  [744] = "0.00,0.00,0.00,90.00,0.00,90.00,0,"
  [745] = "0.00,0.00,0.00,90.00,0.00,90.00,0,"
  [746] = "0.00,0.00,0.00,90.00,0.00,90.00,0,"
  [747] = "0.00,0.00,0.00,90.00,0.00,90.00,1,"
  [748] = "0.00,0.00,0.00,90.00,0.00,90.00,0,"
  [749] = "0.00,0.00,0.00,90.00,0.00,90.00,0,"
  [750] = "0.00,0.00,0.00,90.00,0.00,90.00,0,"
  [751] = "0.00,0.00,0.00,90.00,0.00,90.00,1,"
  [752] = "0.00,0.00,0.00,90.00,0.00,90.00,0,"
  [753] = "0.00,0.00,0.00,90.00,0.00,90.00,0,"
  [754] = "0.00,0.00,0.00,90.00,0.00,90.00,0,"
  [755] = "0.00,0.00,0.00,90.00,0.00,90.00,1,"
  [756] = "0.00,0.00,0.00,90.00,0.00,90.00,0,"
  [757] = "0.00,0.00,0.00,90.00,0.00,90.00,0,"
  [758] = "0.00,0.00,0.00,90.00,0.00,90.00,0,"
  [759] = "0.00,0.00,0.00,90.00,0.00,90.00,1,"
  [760] = "0.00,0.00,0.00,90.00,0.00,90.00,0,"
  [761] = "0.00,0.00,0.00,90.00,0.00,90.00,0,"
  [762] = "0.00,0.00,0.00,90.00,0.00,90.00,0,"
  [763] = "0.00,0.00,0.00,90.00,0.00,90.00,1,"
  [764] = "0.00,0.00,0.00,90.00,0.00,90.00,0,"
  [765] = "0.00,0.00,0.00,90.00,0.00,90.00,0,"
  [766] = "0.00,0.00,0.00,90.00,0.00,90.00,0,"
  [767] = "0.00,0.00,0.00,90.00,0.00,90.00,1,"
  [768] = "0.00,0.00,0.00,90.00,0.00,90.00,0,"
  [769] = "0.00,0.00,0.00,90.00,0.00,90.00,0,"
  [770] = "0.00,0.00,0.00,90.00,0.00,90.00,0,"
  [771] = "0.00,0.00,0.00,90.00,0.00,90.00,1,"
  [772] = "0.00,0.00,0.00,90.00,0.00,90.00,0,"
  [773] = "0.00,0.00,0.00,90.00,0.00,90.00,0,"
  [774] = "0.00,0.00,0.00,90.00,0.00,90.00,0,"
  [775] = "0.00,0.00,0.00,90.00,0.00,90.00,1,"
  [776] = "0.00,0.00,0.00,90.00,0.00,90.00,0,"
  [777] = "0.00,0.00,0.00,90.00,0.00,90.00,0,"
  [778] = "0.00,0.00,0.00,90.00,0.00,90.00,0,"
  [779] = "0.00,0.00,0.00,90.00,0.00,90.00,1,"
  [780] = "0.00,0.00,0.00,90.00,0.00,90.00,0,"
  [781] = "0.00,0.00,0.00,90.00,0.00,90.00,0,"
  [782] = "0.00,0.00,0.00,90.00,0.00,90.00,0,"
  [783] = "0.00,0.00,0.00,90.00,0.00,90.00,1,"
  [784] = "0.00,0.00,0.00,90.00,0.00,90.00,0,"
  [785] = "0.00,0.00,0.00,90.00,0.00,90.00,0,"
  [786] = "0.00,0.00,0.00,90.00,0.00,90.00,0,"
  [787] = "0.00,0.00,0.00,90.00,0.00,90.00,1,"
  [788] = "0.00,0.00,0.00,90.00,0.00,90.00,0,"
  [789] = "0.00,0.00,0.00,90.00,0.00,90.00,0,"
  [790] = "0.00,0.00,0.00,90.00,0.00,90.00,0,"
  [791] = "0.00,0.00,0.00,90.00,0.00,90.00,1,"
  [792] = "0.00,0.00,0.00,90.00,0.00,90.00,0,"
  [793] = "0.00,0.00,0.00,90.00,0.00,90.00,0,"
  [794] = "0.00,0.00,0.00,90.00,0.00,90.00,0,"
  [795] = "0.00,0.00,0.00,90.00,0.00,90.00,1,"
  [796] = "0.00,0.00,0.00,90.00,0.00,90.00,0,"
  [797] = "0.00,0.00,0.00,90.00,0.00,90.00,0,"
  [798] = "0.00,0.00,0.00,90.00,0.00,90.00,0,"
  [799] = "0.00,0.00,0.00,90.00,0.00,90.00,1,"
  [800] = "0.00,0.00,0.00,90.00,0.00,90.00,0,"
  [801] = "0.00,0.00,0.00,90.00,0.00,90.00,0,"
  [802] = "0.00,0.00,0.00,90.00,0.00,90.00,0,"
  [803] = "0.00,0.00,0.00,90.00,0.00,90.00,1,"
  [804] = "0.00,0.00,0.00,90.00,0.00,90.00,0,"
  [805] = "0.00,0.00,0.00,90.00,0.00,90.00,0,"
  [806] = "0.00,0.00,0.00,90.00,0.00,90.00,0,"
  [807] = "0.00,0.00,0.00,90.00,0.00,90.00,1,"
  [808] = "0.00,0.00,0.00,90.00,0.00,90.00,0,"
  [809] = "0.00,0.00,0.00,90.00,0.00,90.00,0,"
  [810] = "0.00,0.00,0.00,90.00,0.00,90.00,0,"
  [811] = "0.00,0.00,0.00,90.00,0.00,90.00,1,"
  [812] = "0.00,0.00,0.00,90.00,0.00,90.00,0,"
  [813] = "0.00,0.00,0.00,90.00,0.00,90.00,0,"
  [814] = "0.00,0.00,0.00,90.00,0.00,90.00,0,"
  [815] = "0.00,0.00,0.00,90.00,0.00,90.00,1,"
  [816] = "0.00,0.00,0.00,90.00,0.00,90.00,0,"
  [817] = "0.00,0.00,0.00,90.00,0.00,90.00,0,"
  [818] = "0.00,0.00,0.00,90.00,0.00,90.00,0,"
  [819] = "0.00,0.00,0.00,90.00,0.00,90.00,1,"
  [820] = "0.00,0.00,0.00,90.00,0.00,90.00,0,"
  [821] = "0.00,0.00,0.00,90.00,0.00,90.00,0,"
  [822] = "0.00,0.00,0.00,90.00,0.00,90.00,0,"
  [823] = "0.00,0.00,0.00,90.00,0.00,90.00,1,"
  [824] = "0.00,0.00,0.00,90.00,0.00,90.00,0,"
  [825] = "0.00,0.00,0.00,90.00,0.00,90.00,0,"
  [826] = "0.00,0.00,0.00,90.00,0.00,90.00,0,"
  [827] = "0.00,0.00,0.00,90.00,0.00,90.00,1,"
  [828] = "0.00,0.00,0.00,90.00,0.00,90.00,0,"
  [829] = "0.00,0.00,0.00,90.00,0.00,90.00,0,"
  [830] = "0.00,0.00,0.00,90.00,0.00,90.00,0,"
  [831] = "0.00,0.00,0.00,90.00,0.00,90.00,1,"
  [832] = "0.00,0.00,0.00,90.00,0.00,90.00,0,"
  [833] = "0.00,0.00,0.00,90.00,0.00,90.00,0,"
  [834] = "0.00,0.00,0.00,90.00,0.00,90.00,0,"
  [835] = "0.00,0.00,0.00,90.00,0.00,90.00,1,"
  [836] = "0.00,0.00,0.00,90.00,0.00,90.00,0,"
  [837] = "0.00,0.00,0.00,90.00,0.00,90.00,0,"
  [838] = "0.00,0.00,0.00,90.00,0.00,90.00,0,"
  [839] = "0.00,0.00,0.00,90.00,0.00,90.00,1,"
  [840] = "0.00,0.00,0.00,90.00,0.00,90.00,0,"
  [841] = "0.00,0.00,0.00,90.00,0.00,90.00,0,"
  [842] = "0.00,0.00,0.00,90.00,0.00,90.00,0,"
  [843] = "0.00,0.00,0.00,90.00,0.00,90.00,1,"
  [844] = "0.00,0.00,0.00,90.00,0.00,90.00,0,"
  [845] = "0.00,0.00,0.00,90.00,0.00,90.00,0,"
  [846] = "0.00,0.00,0.00,90.00,0.00,90.00,0,"
  [847] = "0.00,0.00,0.00,90.00,0.00,90.00,1,"
  [848] = "0.00,0.00,0.00,90.00,0.00,90.00,0,"
  [849] = "0.00,0.00,0.00,90.00,0.00,90.00,0,"
  [850] = "0.00,0.00,0.00,90.00,0.00,90.00,0,"
  [851] = "0.00,0.00,0.00,90.00,0.00,90.00,1,"
  [852] = "0.00,0.00,0.00,90.00,0.00,90.00,0,"
  [853] = "0.00,0.00,0.00,90.00,0.00,90.00,0,"
  [854] = "0.00,0.00,0.00,90.00,0.00,90.00,0,"
  [855] = "0.00,0.00,0.00,90.00,0.00,90.00,1,"
  [856] = "0.00,0.00,0.00,90.00,0.00,90.00,0,"
  [857] = "0.00,0.00,0.00,90.00,0.00,90.00,0,"
  [858] = "0.00,0.00,0.00,90.00,0.00,90.00,0,"
  [859] = "0.00,0.00,0.00,90.00,0.00,90.00,1,"
  [860] = "0.00,0.00,0.00,90.00,0.00,90.00,0,"
  [861] = "0.00,0.00,0.00,90.00,0.00,90.00,0,"
  [862] = "0.00,0.00,0.00,90.00,0.00,90.00,0,"
  [863] = "0.00,0.00,0.00,90.00,0.00,90.00,1,"
  [864] = "0.00,0.00,0.00,90.00,0.00,90.00,0,"
  [865] = "0.00,0.00,0.00,90.00,0.00,90.00,0,"
  [866] = "0.00,0.00,0.00,90.00,0.00,90.00,0,"
  [867] = "0.00,0.00,0.00,90.00,0.00,90.00,1,"
  [868] = "0.00,0.00,0.00,90.00,0.00,90.00,0,"
  [869] = "0.00,0.00,0.00,90.00,0.00,90.00,0,"
  [870] = "0.00,0.00,0.00,90.00,0.00,90.00,0,"
  [871] = "0.00,0.00,0.00,90.00,0.00,90.00,1,"
  [872] = "0.00,0.00,0.00,90.00,0.00,90.00,0,"
  [873] = "0.00,0.00,0.00,90.00,0.00,90.00,0,"
  [874] = "0.00,0.00,0.00,90.00,0.00,90.00,0,"
  [875] = "0.00,0.00,0.00,90.00,0.00,90.00,1,"
  [876] = "0.00,0.00,0.00,90.00,0.00,90.00,0,"
  [877] = "0.00,0.00,0.00,90.00,0.00,90.00,0,"
  [878] = "0.00,0.00,0.00,90.00,0.00,90.00,0,"
  [879] = "0.00,0.00,0.00,90.00,0.00,90.00,1,"
  [880] = "0.00,0.00,0.00,90.00,0.00,90.00,0,"
  [881] = "0.00,0.00,0.00,90.00,0.00,90.00,0,"
  [882] = "0.00,0.00,0.00,90.00,0.00,90.00,0,"
  [883] = "0.00,0.00,0.00,90.00,0.00,90.00,1,"
  [884] = "0.00,0.00,0.00,90.00,0.00,90.00,0,"
  [885] = "0.00,0.00,0.00,90.00,0.00,90.00,0,"
  [886] = "0.00,0.00,0.00,90.00,0.00,90.00,0,"
  [887] = "0.00,0.00,0.00,90.00,0.00,90.00,1,"
  [888] = "0.00,0.00,0.00,90.00,0.00,90.00,0,"
  [889] = "0.00,0.00,0.00,90.00,0.00,90.00,0,"
  [890] = "0.00,0.00,0.00,90.00,0.00,90.00,0,"
  [891] = "0.00,0.00,0.00,90.00,0.00,90.00,1,"
  [892] = "0.00,0.00,0.00,90.00,0.00,90.00,0,"
  [893] = "0.00,0.00,0.00,90.00,0.00,90.00,0,"
  [894] = "0.00,0.00,0.00,90.00,0.00,90.00,0,"
  [895] = "0.00,0.00,0.00,90.00,0.00,90.00,1,"
  [896] = "0.00,0.00,0.00,90.00,0.00,90.00,0,"
  [897] = "0.00,0.00,0.00,90.00,0.00,90.00,0,"
  [898] = "0.00,0.00,0.00,90.00,0.00,90.00,0,"
  [899] = "0.00,0.00,0.00,90.00,0.00,90.00,1,"
  [900] = "0.00,0.00,0.00,90.00,0.00,90.00,0,"
  [901] = "0.00,0.00,0.00,90.00,0.00,90.00,0,"
  [902] = "0.00,0.00,0.00,90.00,0.00,90.00,0,"
  [903] = "0.00,0.00,0.00,90.00,0.00,90.00,1,"
  [904] = "0.00,0.00,0.00,90.00,0.00,90.00,0,"
  [905] = "0.00,0.00,0.00,90.00,0.00,90.00,0,"
  [906] = "0.00,0.00,0.00,90.00,0.00,90.00,0,"
  [907] = "0.00,0.00,0.00,90.00,0.00,90.00,1,"
  [908] = "0.00,0.00,0.00,90.00,0.00,90.00,0,"
  [909] = "0.00,0.00,0.00,90.00,0.00,90.00,0,"
  [910] = "0.00,0.00,0.00,90.00,0.00,90.00,0,"
  [911] = "0.00,0.00,0.00,90.00,0.00,90.00,1,"
  [912] = "0.00,0.00,0.00,90.00,0.00,90.00,0,"
  [913] = "0.00,0.00,0.00,90.00,0.00,90.00,0,"
  [914] = "0.00,0.00,0.00,90.00,0.00,90.00,0,"
  [915] = "0.00,0.00,0.00,90.00,0.00,90.00,1,"
  [916] = "0.00,0.00,0.00,90.00,0.00,90.00,0,"
  [917] = "0.00,0.00,0.00,90.00,0.00,90.00,0,"
  [918] = "0.00,0.00,0.00,90.00,0.00,90.00,0,"
  [919] = "0.00,0.00,0.00,90.00,0.00,90.00,1,"
  [920] = "0.00,0.00,0.00,90.00,0.00,90.00,0,"
  [921] = "0.00,0.00,0.00,90.00,0.00,90.00,0,"
  [922] = "0.00,0.00,0.00,90.00,0.00,90.00,0,"
  [923] = "0.00,0.00,0.00,90.00,0.00,90.00,1,"
  [924] = "0.00,0.00,0.00,90.00,0.00,90.00,0,"
  [925] = "0.00,0.00,0.00,90.00,0.00,90.00,0,"
  [926] = "0.00,0.00,0.00,90.00,0.00,90.00,0,"
  [927] = "0.00,0.00,0.00,90.00,0.00,90.00,1,"
  [928] = "0.00,0.00,0.00,90.00,0.00,90.00,0,"
  [929] = "0.00,0.00,0.00,90.00,0.00,90.00,0,"
  [930] = "0.00,0.00,0.00,90.00,0.00,90.00,0,"
  [931] = "0.00,0.00,0.00,90.00,0.00,90.00,1,"
  [932] = "0.00,0.00,0.00,90.00,0.00,90.00,0,"
  [933] = "0.00,0.00,0.00,90.00,0.00,90.00,0,"
  [934] = "0.00,0.00,0.00,90.00,0.00,90.00,0,"
  [935] = "0.00,0.00,0.00,90.00,0.00,90.00,1,"
  [936] = "0.00,0.00,0.00,90.00,0.00,90.00,0,"
  [937] = "0.00,0.00,0.00,90.00,0.00,90.00,0,"
  [938] = "0.00,0.00,0.00,90.00,0.00,90.00,0,"
  [939] = "0.00,0.00,0.00,90.00,0.00,90.00,1,"
  [940] = "0.00,0.00,0.00,90.00,0.00,90.00,0,"
  [941] = "0.00,0.00,0.00,90.00,0.00,90.00,0,"
  [942] = "0.00,0.00,0.00,90.00,0.00,90.00,0,"
  [943] = "0.00,0.00,0.00,90.00,0.00,90.00,1,"
  [944] = "0.00,0.00,0.00,90.00,0.00,90.00,0,"
  [945] = "0.00,0.00,0.00,90.00,0.00,90.00,0,"
  [946] = "0.00,0.00,0.00,90.00,0.00,90.00,0,"
  [947] = "0.00,0.00,0.00,90.00,0.00,90.00,1,"
  [948] = "0.00,0.00,0.00,90.00,0.00,90.00,0,"
  [949] = "0.00,0.00,0.00,90.00,0.00,90.00,0,"
  [950] = "0.00,0.00,0.00,90.00,0.00,90.00,0,"
  [951] = "0.00,0.00,0.00,90.00,0.00,90.00,1,"
  [952] = "0.00,0.00,0.00,90.00,0.00,90.00,0,"
  [953] = "0.00,0.00,0.00,90.00,0.00,90.00,0,"
  [954] = "0.00,0.00,0.00,90.00,0.00,90.00,0,"
  [955] = "0.00,0.00,0.00,90.00,0.00,90.00,1,"
  [956] = "0.00,0.00,0.00,90.00,0.00,90.00,0,"
  [957] = "0.00,0.00,0.00,90.00,0.00,90.00,0,"
  [958] = "0.00,0.00,0.00,90.00,0.00,90.00,0,"
  [959] = "0.00,0.00,0.00,90.00,0.00,90.00,1,"
  [960] = "0.00,0.00,0.00,90.00,0.00,90.00,0,"
  [961] = "0.00,0.00,0.00,90.00,0.00,90.00,0,"
  [962] = "0.00,0.00,0.00,90.00,0.00,90.00,0,"
  [963] = "0.00,0.00,0.00,90.00,0.00,90.00,1,"
  [964] = "0.00,0.00,0.00,90.00,0.00,90.00,0,"
  [965] = "0.00,0.00,0.00,90.00,0.00,90.00,0,"
  [966] = "0.00,0.00,0.00,90.00,0.00,90.00,0,"
  [967] = "0.00,0.00,0.00,90.00,0.00,90.00,1,"
  [968] = "0.00,0.00,0.00,90.00,0.00,90.00,0,"
  [969] = "0.00,0.00,0.00,90.00,0.00,90.00,0,"
  [970] = "0.00,0.00,0.00,90.00,0.00,90.00,0,"
  [971] = "0.00,0.00,0.00,90.00,0.00,90.00,1,"
  [972] = "0.00,0.00,0.00,90.00,0.00,90.00,0,"
  [973] = "0.00,0.00,0.00,90.00,0.00,90.00,0,"
  [974] = "0.00,0.00,0.00,90.00,0.00,90.00,0,"
  [975] = "0.00,0.00,0.00,90.00,0.00,90.00,1,"
  [976] = "0.00,0.00,0.00,90.00,0.00,90.00,0,"
  [977] = "0.00,0.00,0.00,90.00,0.00,90.00,0,"
  [978] = "0.00,0.00,0.00,90.00,0.00,90.00,0,"
  [979] = "0.00,0.00,0.00,90.00,0.00,90.00,1,"
  [980] = "0.00,0.00,0.00,90.00,0.00,90.00,0,"
  [981] = "0.00,0.00,0.00,90.00,0.00,90.00,0,"
  [982] = "0.00,0.00,0.00,90.00,0.00,90.00,0,"
  [983] = "0.00,0.00,0.00,90.00,0.00,90.00,1,"
  [984] = "0.00,0.00,0.00,90.00,0.00,90.00,0,"
  [985] = "0.00,0.00,0.00,90.00,0.00,90.00,0,"
  [986] = "0.00,0.00,0.00,90.00,0.00,90.00,0,"
  [987] = "0.00,0.00,0.00,90.00,0.00,90.00,1,"
  [988] = "0.00,0.00,0.00,90.00,0.00,90.00,0,"
  [989] = "0.00,0.00,0.00,90.00,0.00,90.00,0,"
  [990] = "0.00,0.00,0.00,90.00,0.00,90.00,0,"
  [991] = "0.00,0.00,0.00,90.00,0.00,90.00,1,"
  [992] = "0.00,0.00,0.00,90.00,0.00,90.00,0,"
  [993] = "0.00,0.00,0.00,90.00,0.00,90.00,0,"
  [994] = "0.00,0.00,0.00,90.00,0.00,90.00,0,"
  [995] = "0.00,0.00,0.00,90.00,0.00,90.00,1,"
  [996] = "0.00,0.00,0.00,90.00,0.00,90.00,0,"
  [997] = "0.00,0.00,0.00,90.00,0.00,90.00,0,"
  [998] = "0.00,0.00,0.00,90.00,0.00,90.00,0,"
  [999] = "0.00,0.00,0.00,90.00,0.00,90.00,1,"
  [1000] = "0.00,0.00,0.00,90.00,0.00,90.00,0,"
  [1001] = "0.00,0.00,0.00,90.00,0.00,90.00,0,"
  [1002] = "0.00,0.00,0.00,90.00,0.00,90.00,0,"
  [1003] = "0.00,0.00,0.00,90.00,0.00,90.00,1,"
  [1004] = "0.00,0.00,0.00,90.00,0.00,90.00,0,"
  [1005] = "0.00,0.00,0.00,90.00,0.00,90.00,0,"
  [1006] = "0.00,0.00,0.00,90.00,0.00,90.00,0,"
  [1007] = "0.00,0.00,0.00,90.00,0.00,90.00,1,"
  [1008] = "0.00,0.00,0.00,90.00,0.00,90.00,0,"
  [1009] = "0.00,0.00,0.00,90.00,0.00,90.00,0,"
  [1010] = "0.00,0.00,0.00,90.00,0.00,90.00,0,"
  [1011] = "0.00,0.00,0.00,90.00,0.00,90.00,1,"
  [1012] = "0.00,0.00,0.00,90.00,0.00,90.00,0,"
  [1013] = "0.00,0.00,0.00,90.00,0.00,90.00,0,"
  [1014] = "0.00,0.00,0.00,90.00,0.00,90.00,0,"
  [1015] = "0.00,0.00,0.00,90.00,0.00,90.00,1,"
  [1016] = "0.00,0.00,0.00,90.00,0.00,90.00,0,"
  [1017] = "0.00,0.00,0.00,90.00,0.00,90.00,0,"
  [1018] = "0.00,0.00,0.00,90.00,0.00,90.00,0,"
  [1019] = "0.00,0.00,0.00,90.00,0.00,90.00,1,"
  [1020] = "0.00,0.00,0.00,90.00,0.00,90.00,0,"
  [1021] = "0.00,0.00,0.00,90.00,0.00,90.00,0,"
  [1022] = "0.00,0.00,0.00,90.00,0.00,90.00,0,"
  [1023] = "0.00,0.00,0.00,90.00,0.00,90.00,1,"
  [1024] = "0.00,0.00,0.00,90.00,0.00,90.00,0,"
  [1025] = "0.00,0.00,0.00,90.00,0.00,90.00,0,"
  [1026] = "0.00,0.00,0.00,90.00,0.00,90.00,0,"
  [1027] = "0.00,0.00,0.00,90.00,0.00,90.00,1,"
  [1028] = "0.00,0.00,0.00,90.00,0.00,90.00,0,"
  [1029] = "0.00,0.00,0.00,90.00,0.00,90.00,0,"
  [1030] = "0.00,0.00,0.00,90.00,0.00,90.00,0,"
  [1031] = "0.00,0.00,0.00,90.00,0.00,90.00,1,"
  [1032] = "0.00,0.00,0.00,90.00,0.00,90.00,0,"
  [1033] = "0.00,0.00,0.00,90.00,0.00,90.00,0,"
  [1034] = "0.00,0.00,0.00,90.00,0.00,90.00,0,"
  [1035] = "0.00,0.00,0.00,90.00,0.00,90.00,1,"
  [1036] = "0.00,0.00,0.00,90.00,0.00,90.00,0,"
  [1037] = "0.00,0.00,0.00,90.00,0.00,90.00,0,"
  [1038] = "0.00,0.00,0.00,90.00,0.00,90.00,0,"
  [1039] = "0.00,0.00,0.00,90.00,0.00,90.00,1,"
  [1040] = "0.00,0.00,0.00,90.00,0.00,90.00,0,"
  [1041] = "0.00,0.00,0.00,90.00,0.00,90.00,0,"
  [1042] = "0.00,0.00,0.00,90.00,0.00,90.00,0,"
  [1043] = "0.00,0.00,0.00,90.00,0.00,90.00,1,"
  [1044] = "0.00,0.00,0.00,90.00,0.00,90.00,0,"
  [1045] = "0.00,0.00,0.00,90.00,0.00,90.00,0,"
  [1046] = "0.00,0.00,0.00,90.00,0.00,90.00,0,"
  [1047] = "0.00,0.00,0.00,90.00,0.00,90.00,1,"
  [1048] = "0.00,0.00,0.00,90.00,0.00,90.00,0,"
  [1049] = "0.00,0.00,0.00,90.00,0.00,90.00,0,"
  [1050] = "0.00,0.00,0.00,90.00,0.00,90.00,0,"
  [1051] = "0.00,0.00,0.00,90.00,0.00,90.00,1,"
  [1052] = "0.00,0.00,0.00,90.00,0.00,90.00,0,"
  [1053] = "0.00,0.00,0.00,90.00,0.00,90.00,0,"
  [1054] = "0.00,0.00,0.00,90.00,0.00,90.00,0,"
  [1055] = "0.00,0.00,0.00,90.00,0.00,90.00,1,"
  [1056] = "0.00,0.00,0.00,90.00,0.00,90.00,0,"
  [1057] = "0.00,0.00,0.00,90.00,0.00,90.00,0,"
  [1058] = "0.00,0.00,0.00,90.00,0.00,90.00,0,"
  [1059] = "0.00,0.00,0.00,90.00,0.00,90.00,1,"
  [1060] = "0.00,0.00,0.00,90.00,0.00,90.00,0,"
  [1061] = "0.00,0.00,0.00,90.00,0.00,90.00,0,"
  [1062] = "0.00,0.00,0.00,90.00,0.00,90.00,0,"
  [1063] = "0.00,0.00,0.00,90.00,0.00,90.00,1,"
  [1064] = "0.00,0.00,0.00,90.00,0.00,90.00,0,"
  [1065] = "0.00,0.00,0.00,90.00,0.00,90.00,0,"
  [1066] = "0.00,0.00,0.00,90.00,0.00,90.00,0,"
  [1067] = "0.00,0.00,0.00,90.00,0.00,90.00,1,"
  [1068] = "0.00,0.00,0.00,90.00,0.00,90.00,0,"
  [1069] = "0.00,0.00,0.00,90.00,0.00,90.00,0,"
  [1070] = "0.00,0.00,0.00,90.00,0.00,90.00,0,"
  [1071] = "0.00,0.00,0.00,90.00,0.00,90.00,1,"
  [1072] = "0.00,0.00,0.00,90.00,0.00,90.00,0,"
  [1073] = "0.00,0.00,0.00,90.00,0.00,90.00,0,"
  [1074] = "0.00,0.00,0.00,90.00,0.00,90.00,0,"
  [1075] = "0.00,0.00,0.00,90.00,0.00,90.00,1,"
  [1076] = "0.00,0.00,0.00,90.00,0.00,90.00,0,"
  [1077] = "0.00,0.00,0.00,90.00,0.00,90.00,0,"
  [1078] = "0.00,0.00,0.00,90.00,0.00,90.00,0,"
  [1079] = "0.00,0.00,0.00,90.00,0.00,90.00,1,"
  [1080] = "0.00,0.00,0.00,90.00,0.00,90.00,0,"
  [1081] = "0.00,0.00,0.00,90.00,0.00,90.00,0,"
  [1082] = "0.00,0.00,0.00,90.00,0.00,90.00,0,"
  [1083] = "0.00,0.00,0.00,90.00,0.00,90.00,1,"
  [1084] = "0.00,0.00,0.00,90.00,0.00,90.00,0,"
  [1085] = "0.00,0.00,0.00,90.00,0.00,90.00,0,"
  [1086] = "0.00,0.00,0.00,90.00,0.00,90.00,0,"
  [1087] = "0.00,0.00,0.00,90.00,0.00,90.00,1,"
  [1088] = "0.00,0.00,0.00,90.00,0.00,90.00,0,"
  [1089] = "0.00,0.00,0.00,90.00,0.00,90.00,0,"
  [1090] = "0.00,0.00,0.00,90.00,0.00,90.00,0,"
  [1091] = "0.00,0.00,0.00,90.00,0.00,90.00,1,"
  [1092] = "0.00,0.00,0.00,90.00,0.00,90.00,0,"
  [1093] = "0.00,0.00,0.00,90.00,0.00,90.00,0,"
  [1094] = "0.00,0.00,0.00,90.00,0.00,90.00,0,"
  [1095] = "0.00,0.00,0.00,90.00,0.00,90.00,1,"
  [1096] = "0.00,0.00,0.00,90.00,0.00,90.00,0,"
  [1097] = "0.00,0.00,0.00,90.00,0.00,90.00,0,"
  [1098] = "0.00,0.00,0.00,90.00,0.00,90.00,0,"
  [1099] = "0.00,0.00,0.00,90.00,0.00,90.00,1,"
  [1100] = "0.00,0.00,0.00,90.00,0.00,90.00,0,"
  [1101] = "0.00,0.00,0.00,90.00,0.00,90.00,0,"
  [1102] = "0.00,0.00,0.00,90.00,0.00,90.00,0,"
  [1103] = "0.00,0.00,0.00,90.00,0.00,90.00,1,"
  [1104] = "0.00,0.00,0.00,90.00,0.00,90.00,0,"
  [1105] = "0.00,0.00,0.00,90.00,0.00,90.00,0,"
  [1106] = "0.00,0.00,0.00,90.00,0.00,90.00,0,"
  [1107] = "0.00,0.00,0.00,90.00,0.00,90.00,1,"
  [1108] = "0.00,0.00,0.00,90.00,0.00,90.00,0,"
  [1109] = "0.00,0.00,0.00,90.00,0.00,90.00,0,"
  [1110] = "0.00,0.00,0.00,90.00,0.00,90.00,0,"
  [1111] = "0.00,0.00,0.00,90.00,0.00,90.00,1,"
  [1112] = "0.00,0.00,0.00,90.00,0.00,90.00,0,"
  [1113] = "0.00,0.00,0.00,90.00,0.00,90.00,0,"
  [1114] = "0.00,0.00,0.00,90.00,0.00,90.00,0,"
  [1115] = "0.00,0.00,0.00,90.00,0.00,90.00,1,"
  [1116] = "0.00,0.00,0.00,90.00,0.00,90.00,0,"
  [1117] = "0.00,0.00,0.00,90.00,0.00,90.00,0,"
  [1118] = "0.00,0.00,0.00,90.00,0.00,90.00,0,"
  [1119] = "0.00,0.00,0.00,90.00,0.00,90.00,1,"
  [1120] = "0.00,0.00,0.00,90.00,0.00,90.00,0,"
  [1121] = "0.00,0.00,0.00,90.00,0.00,90.00,0,"
  [1122] = "0.00,0.00,0.00,90.00,0.00,90.00,0,"
  [1123] = "0.00,0.00,0.00,90.00,0.00,90.00,1,"
  [1124] = "0.00,0.00,0.00,90.00,0.00,90.00,0,"
  [1125] = "0.00,0.00,0.00,90.00,0.00,90.00,0,"
  [1126] = "0.00,0.00,0.00,90.00,0.00,90.00,0,"
  [1127] = "0.00,0.00,0.00,90.00,0.00,90.00,1,"
  [1128] = "0.00,0.00,0.00,90.00,0.00,90.00,0,"
  [1129] = "0.00,0.00,0.00,90.00,0.00,90.00,0,"
  [1130] = "0.00,0.00,0.00,90.00,0.00,90.00,0,"
  [1131] = "0.00,0.00,0.00,90.00,0.00,90.00,1,"
  [1132] = "0.00,0.00,0.00,90.00,0.00,90.00,0,"
  [1133] = "0.00,0.00,0.00,90.00,0.00,90.00,0,"
  [1134] = "0.00,0.00,0.00,90.00,0.00,90.00,0,"
  [1135] = "0.00,0.00,0.00,90.00,0.00,90.00,1,"
  [1136] = "0.00,0.00,0.00,90.00,0.00,90.00,0,"
  [1137] = "0.00,0.00,0.00,90.00,0.00,90.00,0,"
  [1138] = "0.00,0.00,0.00,90.00,0.00,90.00,0,"
  [1139] = "0.00,0.00,0.00,90.00,0.00,90.00,1,"
  [1140] = "0.00,0.00,0.00,90.00,0.00,90.00,0,"
  [1141] = "0.00,0.00,0.00,90.00,0.00,90.00,0,"
  [1142] = "0.00,0.00,0.00,90.00,0.00,90.00,0,"
  [1143] = "0.00,0.00,0.00,90.00,0.00,90.00,1,"
  [1144] = "0.00,0.00,0.00,90.00,0.00,90.00,0,"
  [1145] = "0.00,0.00,0.00,90.00,0.00,90.00,0,"
  [1146] = "0.00,0.00,0.00,90.00,0.00,90.00,0,"
  [1147] = "0.00,0.00,0.00,90.00,0.00,90.00,1,"
  [1148] = "0.00,0.00,0.00,90.00,0.00,90.00,0,"
  [1149] = "0.00,0.00,0.00,90.00,0.00,90.00,0,"
  [1150] = "0.00,0.00,0.00,90.00,0.00,90.00,0,"
  [1151] = "0.00,0.00,0.00,90.00,0.00,90.00,1,"
  [1152] = "0.00,0.00,0.00,90.00,0.00,90.00,0,"
  [1153] = "0.00,0.00,0.00,90.00,0.00,90.00,0,"
  [1154] = "0.00,0.00,0.00,90.00,0.00,90.00,0,"
  [1155] = "0.00,0.00,0.00,90.00,0.00,90.00,1,"
  [1156] = "0.00,0.00,0.00,90.00,0.00,90.00,0,"
  [1157] = "0.00,0.00,0.00,90.00,0.00,90.00,0,"
  [1158] = "0.00,0.00,0.00,90.00,0.00,90.00,0,"
  [1159] = "0.00,0.00,0.00,90.00,0.00,90.00,1,"
  [1160] = "0.00,0.00,0.00,90.00,0.00,90.00,0,"
  [1161] = "0.00,0.00,0.00,90.00,0.00,90.00,0,"
  [1162] = "0.00,0.00,0.00,90.00,0.00,90.00,0,"
  [1163] = "0.00,0.00,0.00,90.00,0.00,90.00,1,"
  [1164] = "0.00,0.00,0.00,90.00,0.00,90.00,0,"
  [1165] = "0.00,0.00,0.00,90.00,0.00,90.00,0,"
  [1166] = "0.00,0.00,0.00,90.00,0.00,90.00,0,"
  [1167] = "0.00,0.00,0.00,90.00,0.00,90.00,1,"
  [1168] = "0.00,0.00,0.00,90.00,0.00,90.00,0,"
  [1169] = "0.00,0.00,0.00,90.00,0.00,90.00,0,"
  [1170] = "0.00,0.00,0.00,90.00,0.00,90.00,0,"
  [1171] = "0.00,0.00,0.00,90.00,0.00,90.00,1,"
  [1172] = "0.00,0.00,0.00,90.00,0.00,90.00,0,"
  [1173] = "0.00,0.00,0.00,90.00,0.00,90.00,0,"
  [1174] = "0.00,0.00,0.00,90.00,0.00,90.00,0,"
  [1175] = "0.00,0.00,0.00,90.00,0.00,90.00,1,"
  [1176] = "0.00,0.00,0.00,90.00,0.00,90.00,0,"
  [1177] = "0.00,0.00,0.00,90.00,0.00,90.00,0,"
  [1178] = "0.00,0.00,0.00,90.00,0.00,90.00,0,"
  [1179] = "0.00,0.00,0.00,90.00,0.00,90.00,1,"
  [1180] = "0.00,0.00,0.00,90.00,0.00,90.00,0,"
  [1181] = "0.00,0.00,0.00,90.00,0.00,90.00,0,"
  [1182] = "0.00,0.00,0.00,90.00,0.00,90.00,0,"
  [1183] = "0.00,0.00,0.00,90.00,0.00,90.00,1,"
  [1184] = "0.00,0.00,0.00,90.00,0.00,90.00,0,"
  [1185] = "0.00,0.00,0.00,90.00,0.00,90.00,0,"
  [1186] = "0.00,0.00,0.00,90.00,0.00,90.00,0,"
  [1187] = "0.00,0.00,0.00,90.00,0.00,90.00,1,"
  [1188] = "0.00,0.00,0.00,90.00,0.00,90.00,0,"
  [1189] = "0.00,0.00,0.00,90.00,0.00,90.00,0,"
  [1190] = "0.00,0.00,0.00,90.00,0.00,90.00,0,"
  [1191] = "0.00,0.00,0.00,90.00,0.00,90.00,1,"
  [1192] = "0.00,0.00,0.00,90.00,0.00,90.00,0,"
  [1193] = "0.00,0.00,0.00,90.00,0.00,90.00,0,"
  [1194] = "0.00,0.00,0.00,90.00,0.00,90.00,0,"
  [1195] = "0.00,0.00,0.00,90.00,0.00,90.00,1,"
  [1196] = "0.00,0.00,0.00,90.00,0.00,90.00,0,"
  [1197] = "0.00,0.00,0.00,90.00,0.00,90.00,0,"
  [1198] = "0.00,0.00,0.00,90.00,0.00,90.00,0,"
  [1199] = "0.00,0.00,0.00,90.00,0.00,90.00,1,"
  [1200] = "0.00,0.00,0.00,90.00,0.00,90.00,0,"
  [1201] = "0.00,0.00,0.00,90.00,0.00,90.00,0,"
  [1202] = "0.00,0.00,0.00,90.00,0.00,90.00,0,"
  [1203] = "0.00,0.00,0.00,90.00,0.00,90.00,1,"
  [1204] = "0.00,0.00,0.00,90.00,0.00,90.00,0,"
  [1205] = "0.00,0.00,0.00,90.00,0.00,90.00,0,"
  [1206] = "0.00,0.00,0.00,90.00,0.00,90.00,0,"
  [1207] = "0.00,0.00,0.00,90.00,0.00,90.00,1,"
  [1208] = "0.00,0.00,0.00,90.00,0.00,90.00,0,"
  [1209] = "0.00,0.00,0.00,90.00,0.00,90.00,0,"
  [1210] = "0.00,0.00,0.00,90.00,0.00,90.00,0,"
  [1211] = "0.00,0.00,0.00,90.00,0.00,90.00,1,"
  [1212] = "0.00,0.00,0.00,90.00,0.00,90.00,0,"
  [1213] = "0.00,0.00,0.00,90.00,0.00,90.00,0,"
  [1214] = "0.00,0.00,0.00,90.00,0.00,90.00,0,"
  [1215] = "0.00,0.00,0.00,90.00,0.00,90.00,1,"
  [1216] = "0.00,0.00,0.00,90.00,0.00,90.00,0,"
  [1217] = "0.00,0.00,0.00,90.00,0.00,90.00,0,"
  [1218] = "0.00,0.00,0.00,90.00,0.00,90.00,0,"
  [1219] = "0.00,0.00,0.00,90.00,0.00,90.00,1,"
  [1220] = "0.00,0.00,0.00,90.00,0.00,90.00,0,"
  [1221] = "0.00,0.00,0.00,90.00,0.00,90.00,0,"
  [1222] = "0.00,0.00,0.00,90.00,0.00,90.00,0,"
  [1223] = "0.00,0.00,0.00,90.00,0.00,90.00,1,"
  [1224] = "0.00,0.00,0.00,90.00,0.00,90.00,0,"
  [1225] = "0.00,0.00,0.00,90.00,0.00,90.00,0,"
  [1226] = "0.00,0.00,0.00,90.00,0.00,90.00,0,"
  [1227] = "0.00,0.00,0.00,90.00,0.00,90.00,1,"
  [1228] = "0.00,0.00,0.00,90.00,0.00,90.00,0,"
  [1229] = "0.00,0.00,0.00,90.00,0.00,90.00,0,"
  [1230] = "0.00,0.00,0.00,90.00,0.00,90.00,0,"
  [1231] = "0.00,0.00,0.00,90.00,0.00,90.00,1,"
  [1232] = "0.00,0.00,0.00,90.00,0.00,90.00,0,"
  [1233] = "0.00,0.00,0.00,90.00,0.00,90.00,0,"
  [1234] = "0.00,0.00,0.00,90.00,0.00,90.00,0,"
  [1235] = "0.00,0.00,0.00,90.00,0.00,90.00,1,"
  [1236] = "0.00,0.00,0.00,90.00,0.00,90.00,0,"
  [1237] = "0.00,0.00,0.00,90.00,0.00,90.00,0,"
  [1238] = "0.00,0.00,0.00,90.00,0.00,90.00,0,"
  [1239] = "0.00,0.00,0.00,90.00,0.00,90.00,1,"
  [1240] = "0.00,0.00,0.00,90.00,0.00,90.00,0,"
  [1241] = "0.00,0.00,0.00,90.00,0.00,90.00,0,"
  [1242] = "0.00,0.00,0.00,90.00,0.00,90.00,0,"
  [1243] = "0.00,0.00,0.00,90.00,0.00,90.00,1,"
  [1244] = "0.00,0.00,0.00,90.00,0.00,90.00,0,"
  [1245] = "0.00,0.00,0.00,90.00,0.00,90.00,0,"
  [1246] = "0.00,0.00,0.00,90.00,0.00,90.00,0,"
  [1247] = "0.00,0.00,0.00,90.00,0.00,90.00,1,"
  [1248] = "0.00,0.00,0.00,90.00,0.00,90.00,0,"
  [1249] = "0.00,0.00,0.00,90.00,0.00,90.00,0,"
  [1250] = "0.00,0.00,0.00,90.00,0.00,90.00,0,"
  [1251] = "0.00,0.00,0.00,90.00,0.00,90.00,1,"
  [1252] = "0.00,0.00,0.00,90.00,0.00,90.00,0,"
  [1253] = "0.00,0.00,0.00,90.00,0.00,90.00,0,"
  [1254] = "0.00,0.00,0.00,90.00,0.00,90.00,0,"
  [1255] = "0.00,0.00,0.00,90.00,0.00,90.00,1,"
  [1256] = "0.00,0.00,0.00,90.00,0.00,90.00,0,"
  [1257] = "0.00,0.00,0.00,90.00,0.00,90.00,0,"
  [1258] = "0.00,0.00,0.00,90.00,0.00,90.00,0,"
  [1259] = "0.00,0.00,0.00,90.00,0.00,90.00,1,"
  [1260] = "0.00,0.00,0.00,90.00,0.00,90.00,0,"
  [1261] = "0.00,0.00,0.00,90.00,0.00,90.00,0,"
  [1262] = "0.00,0.00,0.00,90.00,0.00,90.00,0,"
  [1263] = "0.00,0.00,0.00,90.00,0.00,90.00,1,"
  [1264] = "0.00,0.00,0.00,90.00,0.00,90.00,0,"
  [1265] = "0.00,0.00,0.00,90.00,0.00,90.00,0,"
  [1266] = "0.00,0.00,0.00,90.00,0.00,90.00,0,"
  [1267] = "0.00,0.00,0.00,90.00,0.00,90.00,1,"
  [1268] = "0.00,0.00,0.00,90.00,0.00,90.00,0,"
  [1269] = "0.00,0.00,0.00,90.00,0.00,90.00,0,"
  [1270] = "0.00,0.00,0.00,90.00,0.00,90.00,0,"
  [1271] = "0.00,0.00,0.00,90.00,0.00,90.00,1,"
  [1272] = "0.00,0.00,0.00,90.00,0.00,90.00,0,"
  [1273] = "0.00,0.00,0.00,90.00,0.00,90.00,0,"
  [1274] = "0.00,0.00,0.00,90.00,0.00,90.00,0,"
  [1275] = "0.00,0.00,0.00,90.00,0.00,90.00,1,"
  [1276] = "0.00,0.00,0.00,90.00,0.00,90.00,0,"
  [1277] = "0.00,0.00,0.00,90.00,0.00,90.00,0,"
  [1278] = "0.00,0.00,0.00,90.00,0.00,90.00,0,"
  [1279] = "0.00,0.00,0.00,90.00,0.00,90.00,1,"
  [1280] = "0.00,0.00,0.00,90.00,0.00,90.00,0,"
  [1281] = "0.00,0.00,0.00,90.00,0.00,90.00,0,"
  [1282] = "0.00,0.00,0.00,90.00,0.00,90.00,0,"
  [1283] = "0.00,0.00,0.00,90.00,0.00,90.00,1,"
  [1284] = "0.00,0.00,0.00,90.00,0.00,90.00,0,"
  [1285] = "0.00,0.00,0.00,90.00,0.00,90.00,0,"
  [1286] = "0.00,0.00,0.00,90.00,0.00,90.00,0,"
  [1287] = "0.00,0.00,0.00,90.00,0.00,90.00,1,"
  [1288] = "0.00,0.00,0.00,90.00,0.00,90.00,0,"
  [1289] = "0.00,0.00,0.00,90.00,0.00,90.00,0,"
  [1290] = "0.00,0.00,0.00,90.00,0.00,90.00,0,"
  [1291] = "0.00,0.00,0.00,90.00,0.00,90.00,1,"
  [1292] = "0.00,0.00,0.00,90.00,0.00,90.00,0,"
  [1293] = "0.00,0.00,0.00,90.00,0.00,90.00,0,"
  [1294] = "0.00,0.00,0.00,90.00,0.00,90.00,0,"
  [1295] = "0.00,0.00,0.00,90.00,0.00,90.00,1,"
  [1296] = "0.00,0.00,0.00,90.00,0.00,90.00,0,"
  [1297] = "0.00,0.00,0.00,90.00,0.00,90.00,0,"
  [1298] = "0.00,0.00,0.00,90.00,0.00,90.00,0,"
  [1299] = "0.00,0.00,0.00,90.00,0.00,90.00,1,"
  [1300] = "0.00,0.00,0.00,90.00,0.00,90.00,0,"
  [1301] = "0.00,0.00,0.00,90.00,0.00,90.00,0,"
  [1302] = "0.00,0.00,0.00,90.00,0.00,90.00,0,"
  [1303] = "0.00,0.00,0.00,90.00,0.00,90.00,1,"
  [1304] = "0.00,0.00,0.00,90.00,0.00,90.00,0,"
  [1305] = "0.00,0.00,0.00,90.00,0.00,90.00,0,"
  [1306] = "0.00,0.00,0.00,90.00,0.00,90.00,0,"
  [1307] = "0.00,0.00,0.00,90.00,0.00,90.00,1,"
  [1308] = "0.00,0.00,0.00,90.00,0.00,90.00,0,"
  [1309] = "0.00,0.00,0.00,90.00,0.00,90.00,0,"
  [1310] = "0.00,0.00,0.00,90.00,0.00,90.00,0,"
  [1311] = "0.00,0.00,0.00,90.00,0.00,90.00,1,"
  [1312] = "0.00,0.00,0.00,90.00,0.00,90.00,0,"
  [1313] = "0.00,0.00,0.00,90.00,0.00,90.00,0,"
  [1314] = "0.00,0.00,0.00,90.00,0.00,90.00,0,"
  [1315] = "0.00,0.00,0.00,90.00,0.00,90.00,1,"
  [1316] = "0.00,0.00,0.00,90.00,0.00,90.00,0,"
  [1317] = "0.00,0.00,0.00,90.00,0.00,90.00,0,"
  [1318] = "0.00,0.00,0.00,90.00,0.00,90.00,0,"
  [1319] = "0.00,0.00,0.00,90.00,0.00,90.00,1,"
  [1320] = "0.00,0.00,0.00,90.00,0.00,90.00,0,"
  [1321] = "0.00,0.00,0.00,90.00,0.00,90.00,0,"
  [1322] = "0.00,0.00,0.00,90.00,0.00,90.00,0,"
  [1323] = "0.00,0.00,0.00,90.00,0.00,90.00,1,"
  [1324] = "0.00,0.00,0.00,90.00,0.00,90.00,0,"
  [1325] = "0.00,0.00,0.00,90.00,0.00,90.00,0,"
  [1326] = "0.00,0.00,0.00,90.00,0.00,90.00,0,"
  [1327] = "0.00,0.00,0.00,90.00,0.00,90.00,1,"
  [1328] = "0.00,0.00,0.00,90.00,0.00,90.00,0,"
  [1329] = "0.00,0.00,0.00,90.00,0.00,90.00,0,"
  [1330] = "0.00,0.00,0.00,90.00,0.00,90.00,0,"
  [1331] = "0.00,0.00,0.00,90.00,0.00,90.00,1,"
  [1332] = "0.00,0.00,0.00,90.00,0.00,90.00,0,"
  [1333] = "0.00,0.00,0.00,90.00,0.00,90.00,0,"
  [1334] = "0.00,0.00,0.00,90.00,0.00,90.00,0,"
  [1335] = "0.00,0.00,0.00,90.00,0.00,90.00,1,"
  [1336] = "0.00,0.00,0.00,90.00,0.00,90.00,0,"
  [1337] = "0.00,0.00,0.00,90.00,0.00,90.00,0,"
  [1338] = "0.00,0.00,0.00,90.00,0.00,90.00,0,"
  [1339] = "0.00,0.00,0.00,90.00,0.00,90.00,1,"
  [1340] = "0.00,0.00,0.00,90.00,0.00,90.00,0,"
  [1341] = "0.00,0.00,0.00,90.00,0.00,90.00,0,"
  [1342] = "0.00,0.00,0.00,90.00,0.00,90.00,0,"
  [1343] = "0.00,0.00,0.00,90.00,0.00,90.00,1,"
  [1344] = "0.00,0.00,0.00,90.00,0.00,90.00,0,"
  [1345] = "0.00,0.00,0.00,90.00,0.00,90.00,0,"
  [1346] = "0.00,0.00,0.00,90.00,0.00,90.00,0,"
  [1347] = "0.00,0.00,0.00,90.00,0.00,90.00,1,"
  [1348] = "0.00,0.00,0.00,90.00,0.00,90.00,0,"
  [1349] = "0.00,0.00,0.00,90.00,0.00,90.00,0,"
  [1350] = "0.00,0.00,0.00,90.00,0.00,90.00,0,"
  [1351] = "0.00,0.00,0.00,90.00,0.00,90.00,1,"
  [1352] = "0.00,0.00,0.00,90.00,0.00,90.00,0,"
  [1353] = "0.00,0.00,0.00,90.00,0.00,90.00,0,"
  [1354] = "0.00,0.00,0.00,90.00,0.00,90.00,0,"
  [1355] = "0.00,0.00,0.00,90.00,0.00,90.00,1,"
  [1356] = "0.00,0.00,0.00,90.00,0.00,90.00,0,"
  [1357] = "0.00,0.00,0.00,90.00,0.00,90.00,0,"
  [1358] = "0.00,0.00,0.00,90.00,0.00,90.00,0,"
  [1359] = "0.00,0.00,0.00,90.00,0.00,90.00,1,"
  [1360] = "0.00,0.00,0.00,90.00,0.00,90.00,0,"
  [1361] = "0.00,0.00,0.00,90.00,0.00,90.00,0,"
  [1362] = "0.00,0.00,0.00,90.00,0.00,90.00,0,"
  [1363] = "0.00,0.00,0.00,90.00,0.00,90.00,1,"
  [1364] = "0.00,0.00,0.00,90.00,0.00,90.00,0,"
  [1365] = "0.00,0.00,0.00,90.00,0.00,90.00,0,"
  [1366] = "0.00,0.00,0.00,90.00,0.00,90.00,0,"
  [1367] = "0.00,0.00,0.00,90.00,0.00,90.00,1,"
  [1368] = "0.00,0.00,0.00,90.00,0.00,90.00,0,"
  [1369] = "0.00,0.00,0.00,90.00,0.00,90.00,0,"
  [1370] = "0.00,0.00,0.00,90.00,0.00,90.00,0,"
  [1371] = "0.00,0.00,0.00,90.00,0.00,90.00,1,"
  [1372] = "0.00,0.00,0.00,90.00,0.00,90.00,0,"
  [1373] = "0.00,0.00,0.00,90.00,0.00,90.00,0,"
  [1374] = "0.00,0.00,0.00,90.00,0.00,90.00,0,"
  [1375] = "0.00,0.00,0.00,90.00,0.00,90.00,1,"
  [1376] = "0.00,0.00,0.00,90.00,0.00,90.00,0,"
  [1377] = "0.00,0.00,0.00,90.00,0.00,90.00,0,"
  [1378] = "0.00,0.00,0.00,90.00,0.00,90.00,0,"
  [1379] = "0.00,0.00,0.00,90.00,0.00,90.00,1,"
  [1380] = "0.00,0.00,0.00,90.00,0.00,90.00,0,"
  [1381] = "0.00,0.00,0.00,90.00,0.00,90.00,0,"
  [1382] = "0.00,0.00,0.00,90.00,0.00,90.00,0,"
  [1383] = "0.00,0.00,0.00,90.00,0.00,90.00,1,"
  [1384] = "0.00,0.00,0.00,90.00,0.00,90.00,0,"
  [1385] = "0.00,0.00,0.00,90.00,0.00,90.00,0,"
  [1386] = "0.00,0.00,0.00,90.00,0.00,90.00,0,"
  [1387] = "0.00,0.00,0.00,90.00,0.00,90.00,1,"
  [1388] = "0.00,0.00,0.00,90.00,0.00,90.00,0,"
  [1389] = "0.00,0.00,0.00,90.00,0.00,90.00,0,"
  [1390] = "0.00,0.00,0.00,90.00,0.00,90.00,0,"
  [1391] = "0.00,0.00,0.00,90.00,0.00,90.00,1,"
  [1392] = "0.00,0.00,0.00,90.00,0.00,90.00,0,"
  [1393] = "0.00,0.00,0.00,90.00,0.00,90.00,0,"
  [1394] = "0.00,0.00,0.00,90.00,0.00,90.00,0,"
  [1395] = "0.00,0.00,0.00,90.00,0.00,90.00,1,"
  [1396] = "0.00,0.00,0.00,90.00,0.00,90.00,0,"
  [1397] = "0.00,0.00,0.00,90.00,0.00,90.00,0,"
  [1398] = "0.00,0.00,0.00,90.00,0.00,90.00,0,"
  [1399] = "0.00,0.00,0.00,90.00,0.00,90.00,1,"
  [1400] = "0.00,0.00,0.00,90.00,0.00,90.00,0,"
  [1401] = "0.00,0.00,0.00,90.00,0.00,90.00,0,"
  [1402] = "0.00,0.00,0.00,90.00,0.00,90.00,0,"
  [1403] = "0.00,0.00,0.00,90.00,0.00,90.00,1,"
  [1404] = "0.00,0.00,0.00,90.00,0.00,90.00,0,"
  [1405] = "0.00,0.00,0.00,90.00,0.00,90.00,0,"
  [1406] = "0.00,0.00,0.00,90.00,0.00,90.00,0,"
  [1407] = "0.00,0.00,0.00,90.00,0.00,90.00,1,"
  [1408] = "0.00,0.00,0.00,90.00,0.00,90.00,0,"
  [1409] = "0.00,0.00,0.00,90.00,0.00,90.00,0,"
  [1410] = "0.00,0.00,0.00,90.00,0.00,90.00,0,"
  [1411] = "0.00,0.00,0.00,90.00,0.00,90.00,1,"
  [1412] = "0.00,0.00,0.00,90.00,0.00,90.00,0,"
  [1413] = "0.00,0.00,0.00,90.00,0.00,90.00,0,"
  [1414] = "0.00,0.00,0.00,90.00,0.00,90.00,0,"
  [1415] = "0.00,0.00,0.00,90.00,0.00,90.00,1,"
  [1416] = "0.00,0.00,0.00,90.00,0.00,90.00,0,"
  [1417] = "0.00,0.00,0.00,90.00,0.00,90.00,0,"
  [1418] = "0.00,0.00,0.00,90.00,0.00,90.00,0,"
  [1419] = "0.00,0.00,0.00,90.00,0.00,90.00,1,"
  [1420] = "0.00,0.00,0.00,90.00,0.00,90.00,0,"
  [1421] = "0.00,0.00,0.00,90.00,0.00,90.00,0,"
  [1422] = "0.00,0.00,0.00,90.00,0.00,90.00,0,"
  [1423] = "0.00,0.00,0.00,90.00,0.00,90.00,1,"
  [1424] = "0.00,0.00,0.00,90.00,0.00,90.00,0,"
  [1425] = "0.00,0.00,0.00,90.00,0.00,90.00,0,"
  [1426] = "0.00,0.00,0.00,90.00,0.00,90.00,0,"
  [1427] = "0.00,0.00,0.00,90.00,0.00,90.00,1,"
  [1428] = "0.00,0.00,0.00,90.00,0.00,90.00,0,"
  [1429] = "0.00,0.00,0.00,90.00,0.00,90.00,0,"
  [1430] = "0.00,0.00,0.00,90.00,0.00,90.00,0,"
  [1431] = "0.00,0.00,0.00,90.00,0.00,90.00,1,"
  [1432] = "0.00,0.00,0.00,90.00,0.00,90.00,0,"
  [1433] = "0.00,0.00,0.00,90.00,0.00,90.00,0,"
  [1434] = "0.00,0.00,0.00,90.00,0.00,90.00,0,"
  [1435] = "0.00,0.00,0.00,90.00,0.00,90.00,1,"
  [1436] = "0.00,0.00,0.00,90.00,0.00,90.00,0,"
  [1437] = "0.00,0.00,0.00,90.00,0.00,90.00,0,"
  [1438] = "0.00,0.00,0.00,90.00,0.00,90.00,0,"
  [1439] = "0.00,0.00,0.00,90.00,0.00,90.00,1,"
  [1440] = "0.00,0.00,0.00,90.00,0.00,90.00,0,"
  [1441] = "0.00,0.00,0.00,90.00,0.00,90.00,0,"
  [1442] = "0.00,0.00,0.00,90.00,0.00,90.00,0,"
  [1443] = "0.00,0.00,0.00,90.00,0.00,90.00,1,"
  [1444] = "0.00,0.00,0.00,90.00,0.00,90.00,0,"
  [1445] = "0.00,0.00,0.00,90.00,0.00,90.00,0,"
  [1446] = "0.00,0.00,0.00,90.00,0.00,90.00,0,"
  [1447] = "0.00,0.00,0.00,90.00,0.00,90.00,1,"
  [1448] = "0.00,0.00,0.00,90.00,0.00,90.00,0,"
  [1449] = "0.00,0.00,0.00,90.00,0.00,90.00,0,"
  [1450] = "0.00,0.00,0.00,90.00,0.00,90.00,0,"
  [1451] = "0.00,0.00,0.00,90.00,0.00,90.00,1,"
  [1452] = "0.00,0.00,0.00,90.00,0.00,90.00,0,"
  [1453] = "0.00,0.00,0.00,90.00,0.00,90.00,0,"
  [1454] = "0.00,0.00,0.00,90.00,0.00,90.00,0,"
  [1455] = "0.00,0.00,0.00,90.00,0.00,90.00,1,"
  [1456] = "0.00,0.00,0.00,90.00,0.00,90.00,0,"
  [1457] = "0.00,0.00,0.00,90.00,0.00,90.00,0,"
  [1458] = "0.00,0.00,0.00,90.00,0.00,90.00,0,"
  [1459] = "0.00,0.00,0.00,90.00,0.00,90.00,1,"
  [1460] = "0.00,0.00,0.00,90.00,0.00,90.00,0,"
  [1461] = "0.00,0.00,0.00,90.00,0.00,90.00,0,"
  [1462] = "0.00,0.00,0.00,90.00,0.00,90.00,0,"
  [1463] = "0.00,0.00,0.00,90.00,0.00,90.00,1,"
  [1464] = "0.00,0.00,0.00,90.00,0.00,90.00,0,"
  [1465] = "0.00,0.00,0.00,90.00,0.00,90.00,0,"
  [1466] = "0.00,0.00,0.00,90.00,0.00,90.00,0,"
  [1467] = "0.00,0.00,0.00,90.00,0.00,90.00,1,"
  [1468] = "0.00,0.00,0.00,90.00,0.00,90.00,0,"
  [1469] = "0.00,0.00,0.00,90.00,0.00,90.00,0,"
  [1470] = "0.00,0.00,0.00,90.00,0.00,90.00,0,"
  [1471] = "0.00,0.00,0.00,90.00,0.00,90.00,1,"
  [1472] = "0.00,0.00,0.00,90.00,0.00,90.00,0,"
  [1473] = "0.00,0.00,0.00,90.00,0.00,90.00,0,"
  [1474] = "0.00,0.00,0.00,90.00,0.00,90.00,0,"
  [1475] = "0.00,0.00,0.00,90.00,0.00,90.00,1,"
  [1476] = "0.00,0.00,0.00,90.00,0.00,90.00,0,"
  [1477] = "0.00,0.00,0.00,90.00,0.00,90.00,0,"
  [1478] = "0.00,0.00,0.00,90.00,0.00,90.00,0,"
  [1479] = "0.00,0.00,0.00,90.00,0.00,90.00,1,"
  [1480] = "0.00,0.00,0.00,90.00,0.00,90.00,0,"
  [1481] = "0.00,0.00,0.00,90.00,0.00,90.00,0,"
  [1482] = "0.00,0.00,0.00,90.00,0.00,90.00,0,"
  [1483] = "0.00,0.00,0.00,90.00,0.00,90.00,1,"
  [1484] = "0.00,0.00,0.00,90.00,0.00,90.00,0,"
  [1485] = "0.00,0.00,0.00,90.00,0.00,90.00,0,"
  [1486] = "0.00,0.00,0.00,90.00,0.00,90.00,0,"
  [1487] = "0.00,0.00,0.00,90.00,0.00,90.00,1,"
  [1488] = "0.00,0.00,0.00,90.00,0.00,90.00,0,"
  [1489] = "0.00,0.00,0.00,90.00,0.00,90.00,0,"
  [1490] = "0.00,0.00,0.00,90.00,0.00,90.00,0,"
  [1491] = "0.00,0.00,0.00,90.00,0.00,90.00,1,"
  [1492] = "0.00,0.00,0.00,90.00,0.00,90.00,0,"
  [1493] = "0.00,0.00,0.00,90.00,0.00,90.00,0,"
  [1494] = "0.00,0.00,0.00,90.00,0.00,90.00,0,"
  [1495] = "0.00,0.00,0.00,90.00,0.00,90.00,1,"
  [1496] = "0.00,0.00,0.00,90.00,0.00,90.00,0,"
  [1497] = "0.00,0.00,0.00,90.00,0.00,90.00,0,"
  [1498] = "0.00,0.00,0.00,90.00,0.00,90.00,0,"
  [1499] = "0.00,0.00,0.00,90.00,0.00,90.00,1,"
string strCmd = "RBREDY"
string strScrMsg[8]
  [0] = "F1===>robot1 home or ready"
  [1] = "F2===>robot2 home or ready"
  [2] = "F3===>delete points"
  [3] = "F4===>stop sychron"
  [4] = "F5===>start sychron"
  [5] = "F8===>read txt "
tool tTip = {z=66.95, fatherId=flange[0], ioLink=valve1}
public tool tTool = {z=180, fatherId=flange[0], ioLink=valve1}
trsf trsf_test

--- start.pgx ---
public program start()
begin
  setFrame(frm_ori,frm_x,frm_y,FrmDraw)
  call FC_InitData()
  call initCmdBuf()
  //call stringinit()
  //  waitEndMove()


  //movej(jHome,tTool,mSlow)
  //waitEndMove()
  if taskStatus("tcprec")==-1
    taskCreate "tcprec",90,TcpStrRec:SockRec(datar,ststu)
  endIf
  if taskStatus("CmdManage")==-1
    taskCreate "CmdManage",88,CmdManage()
  endIf
  if taskStatus("CmdDeal")==-1
    taskCreate "CmdDeal",89,CmdDeal()
  endIf
  if taskStatus("nId")==-1
    taskCreate "nId",87,setIOTask()
  endIf
  if taskStatus("CmdTxtReading")==-1
    taskCreate "CmdTxtReading",85,CmdTxtReading()
  endIf
  if taskStatus("CtrlLine")==-1
    taskCreate "CtrlLine",80,CtrlLine()
  endIf
  //    if taskStatus("HMI")==-1
  //    taskCreate "HMI",90,HMI()
  //    endIf
  //
  call HMI()
  //call stringinit()
end

--- CmdDeal.pgx ---
program CmdDeal()
  local num ln_i
  local num ln_total
  local string strX
  local string strY
  local num nPosX
  local num nPosY
  local bool bOk
  local num nPosZ
  local string strZ
  local num local1
  local string strAct
  local num nAct
  local bool bTemp
  local joint jTemp1
begin
  while true
    //deal the command from another robot
    if nReadPt!=nWritePt
      strCmd=mid(CmdBuffer[nReadPt],6,1)

      if strCmd=="RBNEXT"
        TcpStrRec:nCtrl=0
      endIf
      if strCmd=="RBHOME"
        bRb2Home=true
        bRb2Ready=false
      endIf
      if strCmd=="RBREDY"
        popUpMsg("okl")
        bRb2Ready=true
        bRb2Home=false
      endIf
      if strCmd=="RBSTOP"
        bRb2Ready=false
        bRb2Home=false
        bRb2Stop=true
        bRb2Start=false
        bSychronOn=false
      endIf
      if strCmd=="RBSTAT"
        bRb2Home=false
        bRb2Stop=false
        bRb2Start=true
        bSychronOn=true
      endIf
      if strCmd=="RBINIT"
        bRb2InitOk=true
      endIf
      if strCmd=="RBAXI8"
        bRb2AXI8=true
      endIf
      CmdBuffer[nReadPt]=""
      CmdTotal=CmdTotal-1
      nReadPt=nReadPt+1
      if nReadPt>=20
        nReadPt=0
      endIf
    endIf
    delay(0)
  endWhile
end

--- CmdManage.pgx ---
program CmdManage()
begin
  while true
    //add data received into buffer
    if ststu==true and CmdTotal<20
      CmdBuffer[nWritePt]=datar
      CmdTotal=CmdTotal+1
      nWritePt=nWritePt+1
      if nWritePt>=20
        nWritePt=0
      endIf
      //HERE BELOW IS HIGH PRIORITY OF HOMING ROBOT
      datar=""
      ststu=false
    endIf
    delay(0)
  endWhile
end

--- CmdTxtReading.pgx ---
program CmdTxtReading()
begin
  call Txt_initData()
  call txt_PkgInit()
  ////  waitEndMove()
  nCycleTotal=200
  while true
    //if n_sTxt<nTxtTotal and nTxtTotal>2
    if n_Roate<nCycleTotal and nTxtTotal>2
      if bTxt1==true
        call TxtReadRoom1()
      else
      endIf
      if bTxt2==true
        call TxtReadRoom2()
      else
      endIf
      if bTxt3==true
        call TxtReadRoom3()
      else
      endIf
    else
    endIf
    //    nScrPts=n_sTxt
    //    call hmi_refreshmain()
    delay(0)
  endWhile
end

--- CtrlLine.pgx ---
program CtrlLine()
begin

  //Ctrl:nCtrl的含义
  //1：主手回起始点
  //2：从手回起始点
  //3：轨迹点初始化
  //4：同步运动停止
  //5：同步运动开始
  //6：清空点库
  //7：轨迹包初始化
  //8：第八轴

  //...........................

  //51：主手回零完成
  //52：从手回零完成
  //531：初始化完毕
  //532：初始化未进行
  //54：同步运动完成
  //55：同步运动中止
  //56：点库已清空
  //57：轨迹包初始化完毕
  //80：第八轴运动结束
  //.........................


  TcpStrRec:nCtrl=0
  while true
    if TcpStrRec:nCtrl==40
      socket="(RBNEXT)"
      bNextStep=true
      TcpStrRec:nCtrl=0
    endIf
    if TcpStrRec:nCtrl==1
      call F1_r1home()
      TcpStrRec:nCtrl=0
    endIf
    if TcpStrRec:nCtrl==2
      call F2_r2home()
      TcpStrRec:nCtrl=0
    endIf
    if TcpStrRec:nCtrl==3
      socket="(RBPOIN)"
      call txt_PkgInit()
      TcpStrRec:nCtrl=0
    endIf
    if TcpStrRec:nCtrl==4
      call F4_stop()
      TcpStrRec:nCtrl=0
    endIf
    if TcpStrRec:nCtrl==5
      call F5_start()
      TcpStrRec:nCtrl=0
    endIf
    if TcpStrRec:nCtrl==6
      call F6_DELT()
      TcpStrRec:nCtrl=0
    endIf
    if TcpStrRec:nCtrl==7
      call hmi_keyinmain()
      TcpStrRec:nCtrl=0
    endIf
    if TcpStrRec:nCtrl==8
      socket="(RBAXI8)"
      TcpStrRec:nCtrl=0
    endIf
    if bRb2AXI8==true
      TcpStrRec:nFeedback=80
      bRb2AXI8=false
    endIf








  endWhile
end

--- F1_r1home.pgx ---
program F1_r1home()
  local joint l_jTemp1
  local bool l_bTemp
begin

  //robot back to JHome and go to cad:pCad[1]
  //    if bTxtPrSv==false
  //    popUpMsg("请首先对点位文件初始化（按F3“PoIn”）")
  //    else
  if bTxtPrSv==false
    TcpStrRec:nFeedback=532
  else
    if bSychronOn==false
      //    MoveTo.trsf=cad:pCad[0].trsf
      //    //MoveTo.trsf=position(cad:pCad[1],FrmDraw)
      //    //sent fisrt point to another robot
      //    call pointToString(MoveTo,sStrPoints)
      //    //io:socket="(MOVE3M   "+sStrPoints+")"
      //    movej(MoveTo,tTool,mNomSpeed)
      //    //
      //    movej(jCad[0],tTool,mNomSpeed)
      MoveTo.trsf=pfrmCad[0].trsf
      l_bTemp=pointToJoint(tTool,jConfig,MoveTo,l_jTemp1)
      //    $movejSync(jJointRx[l_nCount])
      l_jTemp1.j6=0
      movej(l_jTemp1,tTool,mNomSpeed)
      waitEndMove()
      TcpStrRec:nCtrl=51
    else
      popUpMsg("robot is moving")
    endIf
  endIf


end

--- F2_r2home.pgx ---
program F2_r2home()
begin
  //robot 2 move home position
  socket="(RBREDY)"
  watch(bRb2Ready,10)
  if bRb2Ready==true
    TcpStrRec:nFeedback=52
    //
    popUpMsg("Robot 2 is ready!")
  else
    //popUpMsg("Robot 2 is not ready!")
  endIf
end

--- F4_stop.pgx ---
program F4_stop()
begin
  //stop Synchronous move


  bTxt1=false
  bTxt2=false
  bTxt3=false

  bSychronOn=false
  socket="(RBSTOP)"
  wait(bRb2Stop==true)
  if taskStatus("SychMove")!=-1
    taskKill("SychMove")
    call FC_EndMotion()
    wait(taskStatus("SychMove")==-1)

    //popUpMsg("Sychron stoped")
  endIf
  delay(0.5)
  while size(sString)>1
    $ddel(sString,size(sString)-1)
  endWhile
  while size(pfrmCad)>1
    $ddel(pfrmCad,size(pfrmCad)-1)
  endWhile
  while size(nPulse)>1
    $ddel(nPulse,size(nPulse)-1)
  endWhile
  TcpStrRec:nFeedback=55
  bTxtPrSv=false
  sScrPts="NotReady"
  n_sTxt=0
  call hmi_refreshmain()
end

--- F5_start.pgx ---
public program F5_start()
begin
  //start Synchronous move
  if bTxtPrSv==false
    //    popUpMsg("请首先对点位文件初始化（按F3-PoIn）")
    TcpStrRec:nFeedback=532
  else

    socket="(RBSTAT)"
    delay(0.01)
    nTime=0
    nTestNum=0
    if taskStatus("SychMove")==-1
      taskCreateSync "SychMove",0.004,bRes,sychronMove()
      //taskCreateSync "SychMove",0.008,bRes,sychronRealM()
    else
      popUpMsg("Task is already running")
    endIf
  endIf
  //call sychronMove()
end

--- F6_Axis8.pgx ---
program F6_Axis8()
begin
  call Axis8:onF2Event()
end

--- F6_DELT.pgx ---
program F6_DELT()
begin
  while size(sString)>1
    $ddel(sString,size(sString)-1)
  endWhile
  while size(pfrmCad)>1
    $ddel(pfrmCad,size(pfrmCad)-1)
  endWhile
  while size(nPulse)>1
    $ddel(nPulse,size(nPulse)-1)
  endWhile
  n_sTxt=0
  sScrPts="NotReady"
  call hmi_refreshmain()
  popUpMsg("数据已清空,可以关机")

end

--- FC_EndMotion.pgx ---
program FC_EndMotion()
begin
  //this function is to finish the sychronous motion
  $movejSyncEnd()
end

--- FC_InitData.pgx ---
program FC_InitData()
begin
  //initial data
  cls()
  userPage()
  bRb2Start=false
  bRb2Stop=true
  bRb2Ready=false
  bSychronOn=false
  bRb2Home=false
  bRb2InitOk=false
  bTxt1=false
  bTxt2=false
  bTxt3=false
  call initCmdBuf()
end

--- FC_InitMotion.pgx ---
program FC_InitMotion()
begin
  //this function is goiong to begin synchronous motion
  $movejSyncBegin(mNomSpeed)
end

--- HMI.pgx ---
program HMI()
begin
  //This routine is to is HMI to re-teach points
  call hmi_keyinmain()
end

--- hmi_keyinmain.pgx ---
program hmi_keyinmain()
  local num l_nKeyIn
begin
  //user key interface managementcls()
  gotoxy(2,5)
  put("请输入txt文档总包数。如需修改，选择F7重新进行初始化")
  get(nTxtTotal)
  putln(nTxtTotal)
  sScrPts="NotReady"
  do
    l_nKeyIn=getKey()
    switch l_nKeyIn
      case 271
        call F1_r1home()
      break
      case 272
        call F2_r2home()
      break
      case 273
        call txt_PkgInit()
      break
      case 274
        call F4_stop()
      break
      case 275
        call F5_start()
      break
      case 276
        call F6_Axis8()
      break
      case 277
        call hmi_keyinmain()
      break
      case 278
        //        call txt_rd1()
        cls()
        gotoxy(2,5)
        put("Are you sure to quit ? 'Y' or ESC")
        l_nKeyIn=get()
        if l_nKeyIn==121
          l_nKeyIn=278
        else
          l_nKeyIn=0
        endIf
      break
      case 255
        cls()
        l_nKeyIn=255
      break
    endSwitch
    //refresh hmi screen
    call hmi_refreshmain()
    //monitor production task ,if working mode in remote , start it automatically
  until (l_nKeyIn==255)
end

--- hmi_refreshmain.pgx ---
program hmi_refreshmain()
begin
  //main page key input
  //main page key input
  cls()
  //put screen information
  title("SchronTest==>Master")
  //event log display
  gotoxy(1,1)
  // put("─────────Event───────────")
  put("Menu operation───────────")
  gotoxy(1,2)
  put(strScrMsg[0])
  gotoxy(1,3)
  put(strScrMsg[1])
  gotoxy(1,4)
  put(strScrMsg[2])
  gotoxy(1,5)
  put(strScrMsg[3])
  gotoxy(1,6)
  put(strScrMsg[4])
  gotoxy(1,7)
  put(strScrMsg[5])
  gotoxy(1,8)
  put(strScrMsg[6])
  //  gotoxy(1,9)
  //  put(strScrMsg[7])
  gotoxy(1,9)
  put("Path Load Num")
  gotoxy(23,9)
  put("      ")
  gotoxy(23,9)
  put(n_sTxt)
  gotoxy(1,10)
  put("TxtRoom")
  gotoxy(23,10)
  put("      ")
  gotoxy(23,10)
  put(sScrPts)
  gotoxy(1,11)
  put("TxtPKG Totals")
  gotoxy(23,11)
  put("      ")
  gotoxy(23,11)
  put(nTxtTotal)
  gotoxy(10,1)
  gotoxy(0,13)
  put("RB1H")
  gotoxy(5,13)
  put("RB2H")
  gotoxy(10,13)
  put("PoIn")
  gotoxy(15,13)
  put("STOP")
  gotoxy(20,13)
  put("STAT")
  gotoxy(25,13)
  put("AXIS")
  gotoxy(30,13)
  put("PkNm ")
  gotoxy(35,13)
  put("Exit")
  delay(0.1)
  //recieve key and give actions
end

--- initCmdBuf.pgx ---
program initCmdBuf()
  local num i
begin
  for i=0 to 19
    CmdBuffer[i]=""
  endFor
  CmdTotal=0
  nReadPt=0
  nWritePt=0
  //  setFrame(frm_ori,frm_x,frm_y,FrmDraw)
  jConfig=jHome
  libSave()
end

--- setIOTask.pgx ---
program setIOTask()
  local point l_pHere
  local point l_pPrev
  local num l_nNum
begin
  l_pPrev=here(tTool,FrmDraw)
  l_nNum=0
  while true
    if bSetIO==true
      l_pHere=here(tTool,FrmDraw)
      if distance(l_pPrev,l_pHere)>=1
        //        io:fOut0=false
        //        delay(0)
        //        io:fOut0=true
        l_pPrev=l_pHere
        l_nNum=l_nNum+1
        nIONum=l_nNum
        //        gotoxy(35,11)
        //        put(nIONum)
      endIf
    endIf
    gotoxy(35,11)
    put(nTime)
    delay(0.1)
  endWhile
end

--- stringinit.pgx ---
program stringinit()
  local num i
  local string l_str
begin
  //  for i=0 to 500
  //    $dins(sTxtfile,i)
  //    l_str=toString("1",i)
  //    sTxtfile[i]="path"+l_str+".txt"
  //  endFor
end

--- stringtopoint.pgx ---
program stringtopoint(string x_sString (dimensions=1), num x_nNum (dimensions=1))
  local string l_s
  local bool l_btest
  local num nX
  local num nY
  local num nZ
  local num nA
  local num nB
  local num nC
  local pointRx l_pPointRx
  local trsf tTrsf
  local pointRx pChangeMid1
  local num nP
  local pointRx pChangeMid2
begin
  l_s=x_sString
  l_s=toNum(l_s,nX,l_btest)
  l_s=toNum(l_s,nY,l_btest)
  l_s=toNum(l_s,nZ,l_btest)
  l_s=toNum(l_s,nA,l_btest)
  l_s=toNum(l_s,nB,l_btest)
  l_s=toNum(l_s,nC,l_btest)
  l_s=toNum(l_s,nP,l_btest)
  nPulse[x_nNum]=nP

  pChange.trsf.x=nX
  pChange.trsf.z=nZ
  pChange.trsf.y=nY

  pChangeMid1=compose(pChange,FrmDraw,{0,0,0,nA,0,0})
  pChangeMid2=compose(pChangeMid1,FrmDraw,{0,0,0,0,0,nB})
  pfrmCad[x_nNum]=compose(pChangeMid2,FrmDraw,{0,0,0,nC,0,0})
  //// pfrmCad[x_nNum]=compose(pChange,FrmDraw,{0,0,0,0,0,nB})


  pfrmCad[x_nNum].trsf.x=pChange.trsf.x
  pfrmCad[x_nNum].trsf.z=pChange.trsf.z
  pfrmCad[x_nNum].trsf.y=pChange.trsf.y
  //  pfrmCad[x_nNum].trsf.rx=pChange.trsf.rx
  //    pfrmCad[x_nNum].trsf.rz=pChange.trsf.rz
  //    pfrmCad[x_nNum].trsf.ry=pChange.trsf.ry
  pChange[0].trsf={0,0,0,0,0,0}

end

--- sychronMove.pgx ---
public program sychronMove()
  local bool l_bTemp
  local num l_nCount
  local joint l_jTemp1
  local num l_nTime
begin
  if bTxtPrSv==false
    popUpMsg("请首先对点位文件初始化（按F3“PoIn”）")
  endIf
  call FC_InitMotion()
  l_nCount=0
  n_Roate=0
  nCycleTotal=200
  ////判断机械手什么时间停止
  n_NextCount=0
  ////单程点数
  nNextTotal=9450
  ////补发脉冲数
  nPulseTotal=5
  ////第六轴绝对角度
  nAxisSix=0
  bNextStep=false

  bSetIO=true
  //
  nsumtime=clock()
  //////替换
  do
    if pfrmCad[l_nCount].trsf!={0,0,0,0,0,0}
      /////运动部分/////
      l_nTime=clock()
      MoveTo.trsf=pfrmCad[l_nCount].trsf
      l_bTemp=pointToJoint(tTool,jConfig,MoveTo,l_jTemp1)
      l_jTemp1.j6=nAxisSix
      $movejSync(l_jTemp1)

      if nPulse[l_nCount]==1
        fOut0=true
        fOut0=false
      endIf

      ///////判断什么时间停止
      n_NextCount=n_NextCount+1
      if n_NextCount==2*nNextTotal
        n_NextCount=0
      endIf
      if n_NextCount==nNextTotal
        nPulseCount=0
        while (nPulseCount<nPulseTotal)
          nPulseCount=nPulseCount+1
          fOut0=true
          fOut0=false
          delay(0)
        endWhile
        while bNextStep==false
          //fOut0=true
          //fOut0=false
          delay(0)
        endWhile
      endIf


      //      delay(0)
      /////运动部分/////
      pfrmCad[l_nCount].trsf={0,0,0,0,0,0}
      nPulse=0

      if l_nCount==510
        bTxt1=true
      endIf
      if l_nCount==1010
        bTxt2=true
      endIf
      if l_nCount==10
        bTxt3=true
      endIf
    endIf
    if l_nCount==1499
      l_nCount=0
    else
      l_nCount=l_nCount+1
    endIf
    ////    delay(0)
    l_nTime=clock()-l_nTime
    if l_nTime>nTime
      nTime=l_nTime
      nTestNum=l_nCount
    endIf
    delay(0)
    bNextStep=false
  until pfrmCad[l_nCount].trsf=={0,0,0,0,0,0}

  do

    if l_nCount>0 and l_nCount<500
      l_nCount=500
    endIf

    if 500<l_nCount and l_nCount<1000
      l_nCount=1000
    endIf

    if 1000<l_nCount and l_nCount<1500
      l_nCount=0
    endIf

    ////补发脉冲数
    nPulseCount=0
    while (nPulseCount<nPulseTotal)
      nPulseCount=nPulseCount+1
      fOut0=true
      fOut0=false
      delay(0)
    endWhile
    /////运动暂停
    while (bNextStep==false)
      //fOut0=true
      //fOut0=false
      delay(0)
    endWhile
    bNextStep=false


    do
      if pfrmCad[l_nCount].trsf!={0,0,0,0,0,0}
        /////运动部分/////
        l_nTime=clock()
        MoveTo.trsf=pfrmCad[l_nCount].trsf
        l_bTemp=pointToJoint(tTool,jConfig,MoveTo,l_jTemp1)
        l_jTemp1.j6=nAxisSix
        $movejSync(l_jTemp1)

        if nPulse[l_nCount]==1
          fOut0=true
          fOut0=false
        endIf


        ///////判断什么时间停止
        n_NextCount=n_NextCount+1
        if n_NextCount==2*nNextTotal
          n_NextCount=0
        endIf
        if n_NextCount==nNextTotal

          nPulseCount=0
          while (nPulseCount<nPulseTotal)
            nPulseCount=nPulseCount+1
            fOut0=true
            fOut0=false
            delay(0)
          endWhile
          while bNextStep==false
            // fOut0=true
            // fOut0=false
            delay(0)
          endWhile
        endIf


        //      delay(0)
        /////运动部分/////
        pfrmCad[l_nCount].trsf={0,0,0,0,0,0}
        nPulse=0

        if l_nCount==510
          bTxt1=true
        endIf
        if l_nCount==1010
          bTxt2=true
        endIf
        if l_nCount==10
          bTxt3=true
        endIf
      endIf
      if l_nCount==1499
        l_nCount=0
      else
        l_nCount=l_nCount+1
      endIf
      ////    delay(0)
      l_nTime=clock()-l_nTime
      if l_nTime>nTime
        nTime=l_nTime
        nTestNum=l_nCount
      endIf
      delay(0)
      bNextStep=false
    until pfrmCad[l_nCount].trsf=={0,0,0,0,0,0}

    n_Roate=n_Roate+1
  until n_Roate==nCycleTotal-1

  delay(1)
  bTxt1=false
  bTxt2=false
  bTxt3=false
  while size(sString)>1
    $ddel(sString,size(sString)-1)
  endWhile
  while size(pfrmCad)>1
    $ddel(pfrmCad,size(pfrmCad)-1)
  endWhile
  while size(nPulse)>1
    $ddel(nPulse,size(nPulse)-1)
  endWhile
  ///////////////////////////////////////////////////////////////////////////////////////////////////////////////////
  ///王工缓冲传点原稿
  //  wait(bTest[0]==false and bTest[1]==false)
  //  call FC_InitMotion()
  //  l_nCount=0
  //  bSetIO=true
  //  //
  //  nsumtime=clock()
  //  do
  //    if bTest[0]==false
  //      for l_nCount=0 to size(cad:pCad1)-1
  //        //
  //        if cad:pCad1[l_nCount].trsf!={0,0,0,0,0,0}
  //          l_nTime=clock()
  //          //
  //          MoveTo.trsf=cad:pCad1[l_nCount].trsf
  //          l_bTemp=pointToJoint(tTool,jConfig,MoveTo,l_jTemp1)
  //          $movejSync(l_jTemp1)
  //          //$movejSync(cad:jJointRx[l_nCount])
  //          l_nTime=clock()-l_nTime
  //          if l_nTime>nTime
  //            nTime=l_nTime
  //            nTestNum=l_nCount
  //          endIf
  //          delay(0)
  //          cad:pCad1[l_nCount].trsf={0,0,0,0,0,0}
  //        endIf
  //      endFor
  //      bTest[0]=true
  //    elseIf bTest[1]==false
  //      for l_nCount=0 to size(cad:pCad2)-1
  //        //
  //        if cad:pCad2[l_nCount].trsf!={0,0,0,0,0,0}
  //          l_nTime=clock()
  //          //
  //          MoveTo.trsf=cad:pCad2[l_nCount].trsf
  //          l_bTemp=pointToJoint(tTool,jConfig,MoveTo,l_jTemp1)
  //          $movejSync(l_jTemp1)
  //          //$movejSync(cad:jJointRx[l_nCount])
  //          l_nTime=clock()-l_nTime
  //          if l_nTime>nTime
  //            nTime=l_nTime
  //            nTestNum=l_nCount
  //          endIf
  //          delay(0)
  //          cad:pCad2[l_nCount].trsf={0,0,0,0,0,0}
  //        endIf
  //      endFor
  //      bTest[1]=true
  //    endIf
  //
  //  until (bTest[0]==true and bTest[1]==true and cad:pCad1.trsf=={0,0,0,0,0,0} and cad:pCad2.trsf=={0,0,0,0,0,0})
  ///////////////////////////////////////////////////////////////////////////////////////
  bSetIO=false
  //io:socket="(RBSTOP)"
  call FC_EndMotion()
  TcpStrRec:nFeedback=54
  nsumtime=clock()-nsumtime
  bTxtPrSv=false
  sScrPts="NotReady"
  n_sTxt=0
  call hmi_refreshmain()
  //popUpMsg("move end!")
  //  nScrPts=l_nCount
  //  call hmi_refreshmain()
  bTest=true
end

--- Txt_initData.pgx ---
program Txt_initData()
  local num l_nInit
begin
  while size(sString)>1
    $ddel(sString,size(sString)-1)
  endWhile
  while size(pfrmCad)>1
    $ddel(pfrmCad,size(pfrmCad)-1)
  endWhile
  while size(nPulse)>1
    $ddel(nPulse,size(nPulse)-1)
  endWhile
  pfrmCad[0].trsf={0,0,0,0,0,0}
  sString[0]=""
  nPulse[0]=0
  for l_nInit=1 to 1499
    $dins(sString,l_nInit)
    $dins(pfrmCad,l_nInit)
    $dins(nPulse,l_nInit)
  endFor
  bTxtPrSv=false
  sScrPts="NotReady"
  call hmi_refreshmain()


end

--- txt_PkgInit.pgx ---
program txt_PkgInit()
  local bool l_config
  local joint l_jTemp1
begin
  resetMotion()
  call Txt_initData()


  n_sTxt=0
  call TxtReadRoom1()
  if nTxtTotal>1
    call TxtReadRoom2()
  endIf
  l_config=pointToJoint(tTool,jConfig,pfrmCad[0],jConfig)

  bTxtPrSv=true
  sScrPts="OK"
  call hmi_refreshmain()
end

--- TxtReadRoom1.pgx ---
program TxtReadRoom1()
  local num l_n
  local num l_ntest
  local string sTxtfile
  local string l_str
begin
  bTxt1=false
  delay(0.01)
  l_str=toString("1",n_sTxt)
  sTxtfile="path"+l_str+".txt"
  l_ntest=$fileOpen(sTxtfile,"r")
  for l_n=0 to 499
    $fileGet(l_ntest,sString[l_n],1)
    if sString[l_n]!=""
      call stringtopoint(sString[l_n],l_n)
    else
    endIf
  endFor
  delay(0.01)

  call hmi_refreshmain()

  if n_sTxt==nTxtTotal-1
    n_sTxt=0
  else
    n_sTxt=n_sTxt+1
  endIf

  $fileClose(l_ntest)
end

--- TxtReadRoom2.pgx ---
program TxtReadRoom2()
  local num l_n
  local num l_ntest
  local string l_str
  local string sTxtfile
begin
  bTxt2=false
  delay(0.01)
  l_str=toString("1",n_sTxt)
  sTxtfile="path"+l_str+".txt"
  l_ntest=$fileOpen(sTxtfile,"r")
  for l_n=500 to 999
    $fileGet(l_ntest,sString[l_n],1)
    if sString[l_n]!=""
      call stringtopoint(sString[l_n],l_n)
    else
    endIf
  endFor
  delay(0.01)

  call hmi_refreshmain()

  if n_sTxt==nTxtTotal-1
    n_sTxt=0
  else
    n_sTxt=n_sTxt+1
  endIf

  $fileClose(l_ntest)
end

--- TxtReadRoom3.pgx ---
program TxtReadRoom3()
  local num l_ntest
  local num l_n
  local string l_str
  local string sTxtfile
begin
  bTxt3=false
  delay(0.01)
  l_str=toString("1",n_sTxt)
  sTxtfile="path"+l_str+".txt"
  l_ntest=$fileOpen(sTxtfile,"r")
  for l_n=1000 to 1499
    $fileGet(l_ntest,sString[l_n],1)
    if sString[l_n]!=""
      call stringtopoint(sString[l_n],l_n)
    else
    endIf
  endFor
  delay(0.01)


  if n_sTxt==nTxtTotal-1
    n_sTxt=0
  else
    n_sTxt=n_sTxt+1
  endIf

  call hmi_refreshmain()
  $fileClose(l_ntest)
end
